FUNCTION_BLOCK E_DEMUX8 (* Event demultiplexor 8 Events *)
  (* Standard: 61499-1 Annex A; Description: Copyright (c) 2017 fortiss GmbH This program and the accompanying materials are made available under the terms of the Eclipse Public License 2.0 which is available at https://www.eclipse.org/legal/epl-2.0/ SPDX-License-Identifier: EPL-2.0 *)
  (* Version 1.0, 2017-09-22, Alois Zoitl, fortiss GmbH, initial API and implementation and/or initial documentation *)
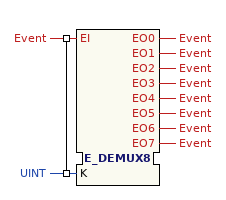
  EVENT_INPUT
    EI WITH K; (* Event to demultiplex *)
  END_EVENT
  EVENT_OUTPUT
    EO0;
    EO1;
    EO2;
    EO3;
    EO4;
    EO5;
    EO6;
    EO7;
  END_EVENT
  VAR_INPUT
    K : UINT; (* Event index *)
  END_VAR
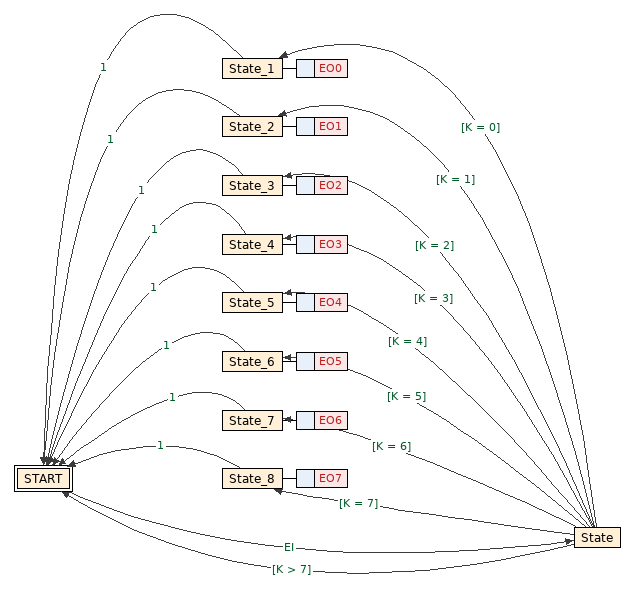
  EC_STATES
    START; (* Initial State *)
    State;
    State_1 : -> EO0;
    State_2 : -> EO1;
    State_3 : -> EO2;
    State_4 : -> EO3;
    State_5 : -> EO4;
    State_6 : -> EO5;
    State_7 : -> EO6;
    State_8 : -> EO7;
  END_STATES
  EC_TRANSITIONS
    State_1 TO START := 1;
    State_2 TO START := 1;
    State_3 TO START := 1;
    State_4 TO START := 1;
    START TO State := EI;
    State TO State_1 := [K = 0];
    State TO State_2 := [K = 1];
    State TO State_3 := [K = 2];
    State TO State_4 := [K = 3];
    State TO State_5 := [K = 4];
    State TO State_6 := [K = 5];
    State TO State_7 := [K = 6];
    State TO State_8 := [K = 7];
    State TO START := [K > 7];
    State_5 TO START := 1;
    State_6 TO START := 1;
    State_7 TO START := 1;
    State_8 TO START := 1;
  END_TRANSITIONS
END_FUNCTION_BLOCK
